(* PLC project Sem nome, Desconhecido Sem nome 1 *)
(* stored: creationDateTime 2019-12-07T15:51:31, modificationDateTime 2019-12-10T18:25:25 *)

PROGRAM Planta
  VAR
    PID0 : PID;
  END_VAR
  VAR
    Setpoint AT %QW1 : INT;
    EN_PID AT %QX0.3 : BOOL;
    KP AT %QW2 : INT;
    TR AT %QW3 : INT;
    TD AT %QW4 : INT;
    VP AT %IW100 : INT;
    SC AT %QW101 : INT;
    QUO AT %QW5 : INT;
  END_VAR

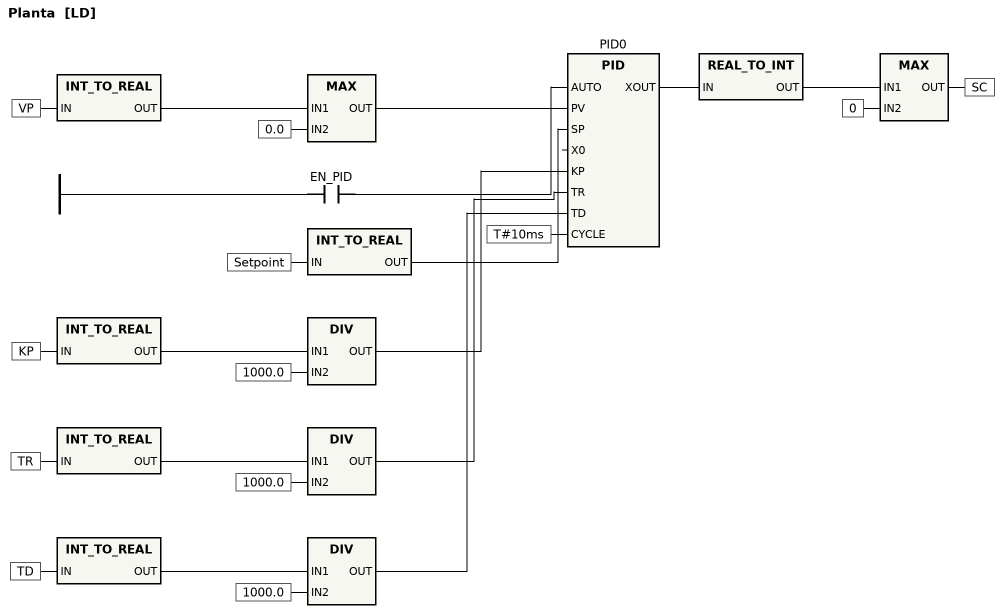
(* LD diagram, written out as Structured Text *)
PID0(AUTO := EN_PID, PV := MAX(INT_TO_REAL(VP), 0.0), SP := INT_TO_REAL(Setpoint), KP := INT_TO_REAL(KP) / 1000.0, TR := INT_TO_REAL(TR) / 1000.0, TD := INT_TO_REAL(TD) / 1000.0, CYCLE := T#10ms);
SC := MAX(REAL_TO_INT(PID0.XOUT), 0);
END_PROGRAM

CONFIGURATION Config0
  RESOURCE Res0 ON PLC
    TASK task0(INTERVAL := T#20ms, PRIORITY := 0);
    PROGRAM instance0 WITH task0 : Planta;
  END_RESOURCE
END_CONFIGURATION
